PROGRAM Q2_MOTOR
VAR
	ClearFault: FB_ClearFault;
	SetEnableState: FB_SetEnableState;
	SetHomingParameter: FB_SetHomingParameter;
	FindHome: FB_FindHome;
	SetMotorParameter: FB_SetMotorParameter;
	SetPositionProfile: FB_SetPositionProfile;
	SetOperationMode: FB_SetOperationMode;
	MoveToPosition: FB_MoveToPosition;
	GetMovementState: FB_GetMovementState;
	SetDisableState: FB_SetDisableState;
	SetPositionMust: FB_SetPositionMust;
	POSITION: DINT;
END_VAR

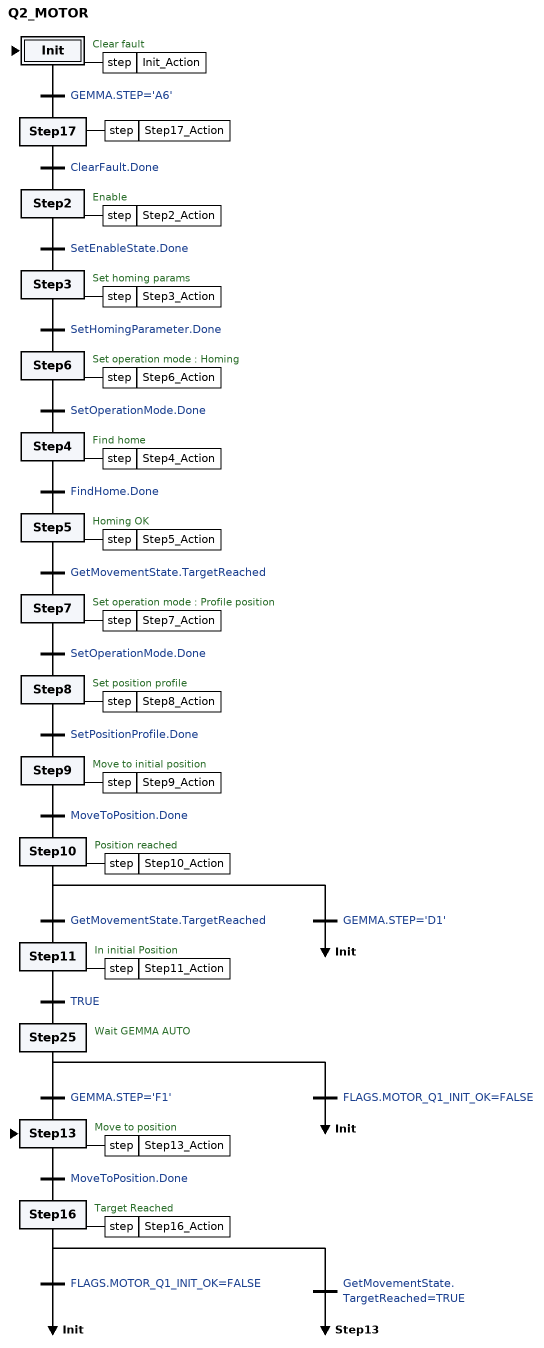
// Clear fault
INITIAL_STEP Init:
    Init_Action(N);  // step action
END_STEP
TRANSITION FROM Init TO Step17
    := GEMMA.STEP='A6';
END_TRANSITION
STEP Step17:
    Step17_Action(N);  // step action
END_STEP
TRANSITION FROM Step17 TO Step2
    := ClearFault.Done;
END_TRANSITION
// Enable
STEP Step2:
    Step2_Action(N);  // step action
END_STEP
TRANSITION FROM Step2 TO Step3
    := SetEnableState.Done;
END_TRANSITION
// Set homing params
STEP Step3:
    Step3_Action(N);  // step action
END_STEP
TRANSITION FROM Step3 TO Step6
    := SetHomingParameter.Done;
END_TRANSITION
// Set operation mode : Homing
STEP Step6:
    Step6_Action(N);  // step action
END_STEP
TRANSITION FROM Step6 TO Step4
    := SetOperationMode.Done;
END_TRANSITION
// Find home
STEP Step4:
    Step4_Action(N);  // step action
END_STEP
TRANSITION FROM Step4 TO Step5
    := FindHome.Done;
END_TRANSITION
// Homing OK
STEP Step5:
    Step5_Action(N);  // step action
END_STEP
TRANSITION FROM Step5 TO Step7
    := GetMovementState.TargetReached;
END_TRANSITION
// Set operation mode : Profile position
STEP Step7:
    Step7_Action(N);  // step action
END_STEP
TRANSITION FROM Step7 TO Step8
    := SetOperationMode.Done;
END_TRANSITION
// Set position profile
STEP Step8:
    Step8_Action(N);  // step action
END_STEP
TRANSITION FROM Step8 TO Step9
    := SetPositionProfile.Done;
END_TRANSITION
// Move to initial position
STEP Step9:
    Step9_Action(N);  // step action
END_STEP
TRANSITION FROM Step9 TO Step10
    := MoveToPosition.Done;
END_TRANSITION
// Position reached
STEP Step10:
    Step10_Action(N);  // step action
END_STEP
TRANSITION FROM Step10 TO Step11
    := GetMovementState.TargetReached;
END_TRANSITION
TRANSITION FROM Step10 TO Init
    := GEMMA.STEP='D1';
END_TRANSITION
// In initial Position
STEP Step11:
    Step11_Action(N);  // step action
END_STEP
TRANSITION FROM Step11 TO Step25
    := TRUE;
END_TRANSITION
// Wait GEMMA AUTO
STEP Step25:
END_STEP
TRANSITION FROM Step25 TO Step13
    := GEMMA.STEP='F1';
END_TRANSITION
TRANSITION FROM Step25 TO Init
    := FLAGS.MOTOR_Q1_INIT_OK=FALSE;
END_TRANSITION
// Move to position
STEP Step13:
    Step13_Action(N);  // step action
END_STEP
TRANSITION FROM Step13 TO Step16
    := MoveToPosition.Done;
END_TRANSITION
// Target Reached
STEP Step16:
    Step16_Action(N);  // step action
END_STEP
TRANSITION FROM Step16 TO Init
    := FLAGS.MOTOR_Q1_INIT_OK=FALSE;
END_TRANSITION
TRANSITION FROM Step16 TO Step13
    := GetMovementState.TargetReached=TRUE;
END_TRANSITION

ACTION Step17_Action:
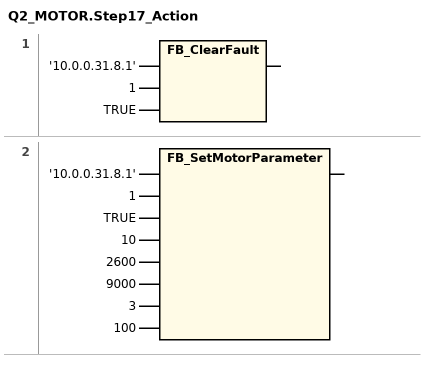
// NETWORK 1
FB_ClearFault('10.0.0.31.8.1', 1, TRUE);

// NETWORK 2
FB_SetMotorParameter('10.0.0.31.8.1', 1, TRUE, 10, 2600, 9000, 3, 100);
END_ACTION

ACTION Step4_Action:
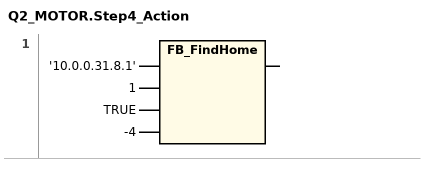
// NETWORK 1
FB_FindHome('10.0.0.31.8.1', 1, TRUE, -4);
END_ACTION

ACTION Step2_Action:
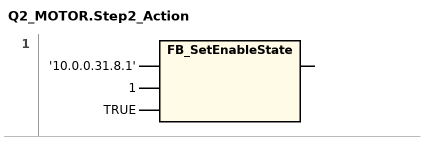
// NETWORK 1
FB_SetEnableState('10.0.0.31.8.1', 1, TRUE);
END_ACTION

ACTION Step13_Action:
(*Limitation deplacement Moteur*)
IF FLAGS.MOTOR_Q2_POSITION>MOTOR_Q2_POSITION_MAX THEN
	POSITION:=MOTOR_Q2_POSITION_MAX;
ELSIF FLAGS.MOTOR_Q2_POSITION<0 THEN
	POSITION:=0;
ELSE
	POSITION:=FLAGS.MOTOR_Q2_POSITION;
END_IF


MoveToPosition(
	ADSNetId:= '10.0.0.31.8.1',
	NodeId:= 1,
	Write:= TRUE,
	TargetPosition:= POSITION,
	Absolut:= TRUE);
END_ACTION

ACTION Step10_Action:
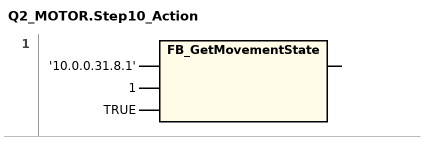
// NETWORK 1
FB_GetMovementState('10.0.0.31.8.1', 1, TRUE);
END_ACTION

ACTION Step5_Action:
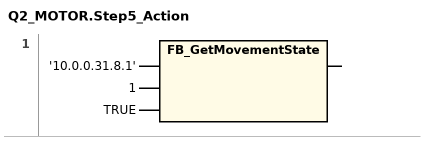
// NETWORK 1
FB_GetMovementState('10.0.0.31.8.1', 1, TRUE);
END_ACTION

ACTION Step7_Action:
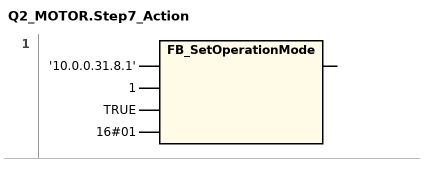
// NETWORK 1
FB_SetOperationMode('10.0.0.31.8.1', 1, TRUE, 16#01);
END_ACTION

ACTION Step9_Action:
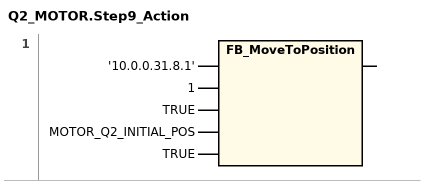
// NETWORK 1
FB_MoveToPosition('10.0.0.31.8.1', 1, TRUE, MOTOR_Q2_INITIAL_POS, TRUE);
END_ACTION

ACTION Step11_Action:

(*SetDisableState(
	ADSNetId:= '10.0.0.31.6.1',
	NodeId:= 1,
	Write:= TRUE);*)

FLAGS.MOTOR_Q2_INIT_OK:=TRUE;
END_ACTION

ACTION Step3_Action:
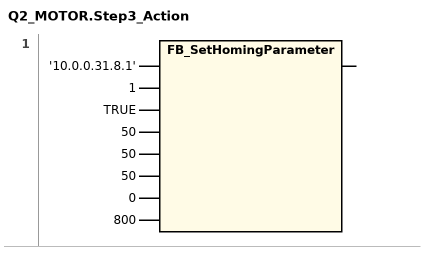
// NETWORK 1
FB_SetHomingParameter('10.0.0.31.8.1', 1, TRUE, 50, 50, 50, 0, 800);
END_ACTION

ACTION Step6_Action:
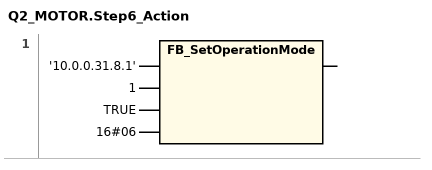
// NETWORK 1
FB_SetOperationMode('10.0.0.31.8.1', 1, TRUE, 16#06);
END_ACTION

ACTION Init_Action:

END_ACTION

ACTION Step16_Action:
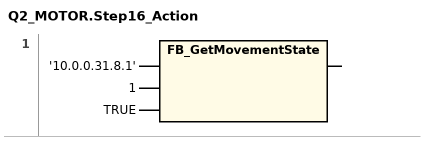
// NETWORK 1
FB_GetMovementState('10.0.0.31.8.1', 1, TRUE);
END_ACTION

ACTION Step8_Action:
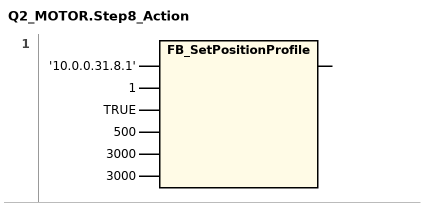
// NETWORK 1
FB_SetPositionProfile('10.0.0.31.8.1', 1, TRUE, 500, 3000, 3000);
END_ACTION

END_PROGRAM

(* stored: Version 1.1.0.1, ProductVersion 3.1.0.26
   POU Q2_MOTOR: Id {0f2aedf8-f292-4ba0-9498-4e6d2da9995a}
   Action Step17_Action: Id {0f461b54-58e6-4a38-9267-c7c6790d4998}
   Action Step4_Action: Id {3154c373-cfd1-4e58-8e35-a8ddd53ec387}
   Action Step2_Action: Id {4383b33e-9cfe-4728-a290-88e8883eb65d}
   Action Step13_Action: Id {4b02d372-06ea-4363-9d35-093a347b6e1a}
   Action Step10_Action: Id {5520bdb4-2da3-43aa-8292-0807edb73356}
   Action Step5_Action: Id {617343bc-2c41-406f-9bda-ddb00283f7cb}
   Action Step7_Action: Id {79d29c08-8e57-49d7-b34e-7b904dd05412}
   Action Step9_Action: Id {885b681f-f260-4f8b-b6c0-c5d2ddcf3ad8}
   Action Step11_Action: Id {a38c4b1b-88ff-4083-9bf5-ac1cd233ae68}
   Action Step3_Action: Id {cb9fafd4-89d7-4330-8f62-537b37b22fdb}
   Action Step6_Action: Id {cea0f7f9-8101-41ea-8278-c531d3cef9bb}
   Action Init_Action: Id {dfed86f3-7a5b-4724-a67e-ef6dd1993e54}
   Action Step16_Action: Id {fac78da0-79c0-4983-8ef7-48a3835817eb}
   Action Step8_Action: Id {fc6e7903-f0d8-4688-97d6-6a858ca73e39} *)
